FUNCTION_BLOCK FB_Robot


VAR_INPUT

END_VAR
VAR_OUTPUT
	bDone: BOOL;
END_VAR
VAR
END_VAR

METHOD AddMission : BOOL
VAR_INPUT
	m: WSTRING;
END_VAR
END_METHOD

METHOD CallSkill : BOOL
VAR_INPUT
	name: WSTRING;
END_VAR
END_METHOD

END_FUNCTION_BLOCK

(* stored: Version 1.1.0.1, ProductVersion 3.1.4026.18
   POU FB_Robot: Id {d67508e2-0ef8-408d-a316-43ebc0a423f1}, SpecialFunc None
   Method AddMission: Id {2710e6d5-8861-49be-b3e5-ece1c90a6c11}
   Method CallSkill: Id {fe5baacd-3adb-45ec-ab40-505efef2d269} *)
